(* PLC project Unnamed, Unknown Unnamed 1 *)
(* stored: creationDateTime 2023-03-26T05:36:49, modificationDateTime 2023-03-26T13:36:35 *)

PROGRAM digdisply
  VAR
    START AT %IX100.0 : BOOL;
    RESET AT %IX100.1 : BOOL;
    Q AT %QX100.0 : BOOL;
    SYSRUN AT %QX0.0 : BOOL;
    DIGDISPY AT %QW100 : INT;
  END_VAR
  VAR
    CTU_DINT0 : CTU_DINT;
  END_VAR
  VAR  (* added by the conversion: wires and edge detectors of the diagram *)
    R_TRIG1 : R_TRIG;
  END_VAR

(* LD diagram, written out as Structured Text *)
SYSRUN := START;
R_TRIG1(CLK := SYSRUN);
CTU_DINT0(CU := R_TRIG1.Q, R := RESET, PV := 5);
Q := CTU_DINT0.Q;
DIGDISPY := DINT_TO_INT(CTU_DINT0.CV);
END_PROGRAM

CONFIGURATION Config0
  RESOURCE Res0 ON PLC
    TASK task0(INTERVAL := T#20ms, PRIORITY := 0);
    PROGRAM instance0 WITH task0 : digdisply;
  END_RESOURCE
END_CONFIGURATION
